TYPE ST_DS402_CSP_Config :
STRUCT	
	fPositionOffset			: LREAL := 0.0;	
	bSwapProcessData		: BOOL; //SWAP Process Data from/to FIELDBUS
END_STRUCT
END_TYPE

(* stored: Version 1.1.0.1, ProductVersion 3.1.4024.12
   DUT ST_DS402_CSP_Config: Id {f0920dfb-66da-09df-2181-42a4491a31ab} *)
